Staubli VAL3: setPalletData.pgx

public program setPalletData(TrajPallet& x_tTrajPallet)
  local num i
begin
  // set the Pallet DATA
  pEditPoint=x_tTrajPallet
  // link it
  for i=0 to size(pEditPoint.tData)-1
    link(pEditPoint.tData[i].pPoint,pEditPoint.fFrame)
  endFor
end
